// LS Electric XG5000 project: CTR
// PLC LSPLC
// module base 0 slot 0: 입출력 모듈:XBC-DR30S (DC 24V 입력 18점, 릴레이 출력 12점)

PROGRAM CTR (task: 스캔 프로그램)

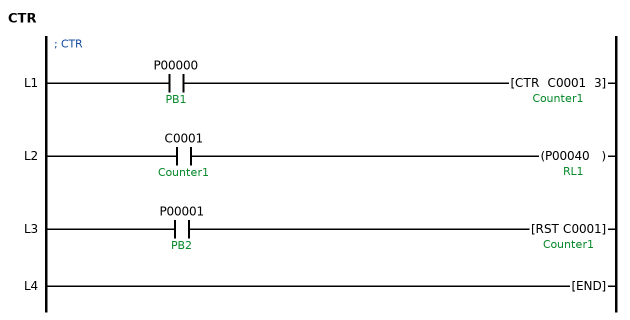
// CTR
; L1
LOAD      P00000	// PB1
CTR       C0001 3	// Counter1
; L2
LOAD      C0001	// Counter1
OUT       P00040	// RL1
; L3
LOAD      P00001	// PB2
RST       C0001	// Counter1
; L4
END